// TIA Portal V20 export
TYPE "LKinCtrl_PathEditor_typeExternalEvents"
// stored: Access Published
   STRUCT
      approachPoint { ExternalAccessible := 'False'; ExternalVisible := 'False'; ExternalWritable := 'False'} : Struct
         trigger : Bool;   // triggers event. Reset internally.
         point : "LKinCtrl_typePoint";   // Selected index in table. Only valid if noSelection = FALSE. / point to approach
      END_STRUCT;
      openTeachKinematics { ExternalAccessible := 'False'; ExternalVisible := 'False'; ExternalWritable := 'False'} : Bool;
      selectedCommandChanged { ExternalAccessible := 'False'; ExternalVisible := 'False'; ExternalWritable := 'False'} : Struct
         trigger : Bool;
         command : "LKinCtrl_typePathDataElement";
      END_STRUCT;
   END_STRUCT;
END_TYPE
